TYPE ST_Values_Energy_Surstoffi :
STRUCT
	sTimestamp			: STRING(255);						//Timestamp
	sID					: STRING(255);						//Id from the Datapoint
	lrValue				: LREAL;							//Value from the Datapoint
END_STRUCT
END_TYPE

(* stored: Version 1.1.0.1, ProductVersion 3.1.4024.9
   DUT ST_Values_Energy_Surstoffi: Id {5a208dd1-8f50-4e36-8348-4049aa098caa} *)
